FUNCTION F_Concat5 : T_MaxString
VAR_INPUT
	sOne : STRING;
	sTwo : STRING;
	sThree : STRING;
	sFour : STRING;
	sFive : STRING;
END_VAR

F_Concat5 := CONCAT(
					sOne,
					F_Concat4( sTwo, sThree, sFour, sFive )
				);

END_FUNCTION

(* stored: Version 1.1.0.1, ProductVersion 3.1.4022.9
   POU F_Concat5: Id {c4214e05-45b2-4d5c-bfe6-cf52d2c16559}, SpecialFunc None *)
